(* PLC project TestPLC, Beckhoff Automation GmbH TwinCAT PLC Control 3.5.8.40 *)
(* stored: creationDateTime 2018-01-04T13:56:45.3224157, modificationDateTime 2018-01-04T13:56:45.3224157 *)

(* global variable list Labview *)
{attribute 'Tc2GvlVarNames'}
{attribute 'TcContextName':='PlcTaskStandard'}
VAR_GLOBAL	
	
(*
	gui_ErrorMessages				:DINT;
	gui_Acknowledge					:BOOL;
	gui_ZustandMaschine				:INT;		(*0: Initialisierung, 1: Stopp, aber alles OK, 2: Produktion automatisch, 3: Schrittbetrieb, 4: Fehler, 5: Manuellbetrieb, 6: Notaus gedrückt, *)
	gui_UserLevel					:INT;		(*Opérateur, Réglage, Maintenance*)
	gui_UserLevelKeySwitchOn		:BOOL;		(*TRUE, wenn Schlüssel auf Service gedreht ist*)
	gui_AktPosAchseZ				:REAL;
	*)
	gui_Play						:BOOL;			
	gui_Stop						:BOOL;		
	gui_Skipback					:BOOL;
	gui_Skipforward					:BOOL;
	gui_Rack						:INT;
	gui_Side						:BOOL;
	gui_Song						:INT;
	gui_Mute						:BOOL;
	gui_IncreaseVolume				:BOOL;
	gui_DecreaseVolume				:BOOL;
	gui_ActRack						:INT;
	gui_ActSide						:BOOL;
	gui_ActSong						:INT;
	
END_VAR
